Staubli VAL3: call.pjx

--- call.pjx ---
Parameters version=s7.2.1 stackSize=5000 millimeterUnit=true
Program file=start.pgx
Program file=stop.pgx
Data file=call.dtx
Library alias=io path=Disk://io/io.pjx

--- call.dtx ---
mdesc nom_speed = {rmax=9999, blend=off}

--- start.pgx ---
public program start()
begin
end

--- stop.pgx ---
program stop()
begin
  popUpMsg("Pending movement commands have been canceled")
  resetMotion()
end
